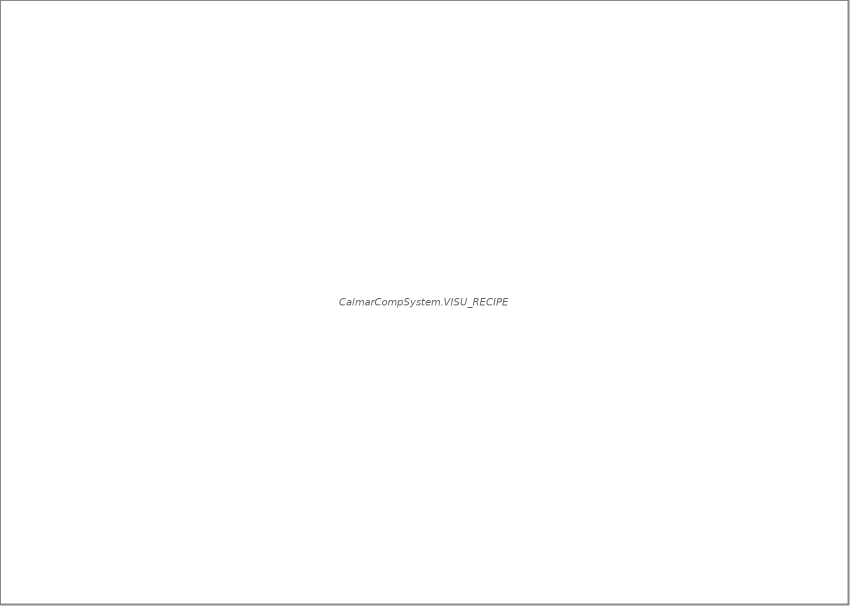
VISUALIZATION VISU_RECIPE  // 850x606
    Frame (0,0 848x604)
        shows CalmarCompSystem.VISU_RECIPE()
END_VISUALIZATION

(* stored: Version 1.1.0.1, ProductVersion 3.1.4024.9
   Visu VISU_RECIPE: Id {5b58c71d-3edb-41d6-9d71-490dd4a04d15} *)
